KUKA KRL program: hmi.src, hmi.dat

--- hmi.src ---
&ACCESS RVO
&REL 6
&PARAM EDITMASK = *
&PARAM TEMPLATE = C:\KRC\Roboter\Template\ExpertVorgabe
DEF hmi( )
wait sec 1000
END

--- hmi.dat ---
&ACCESS RVO
&REL 6
&PARAM EDITMASK = *
&PARAM TEMPLATE = C:\KRC\Roboter\Template\ExpertVorgabe
DEFDAT hmi PUBLIC

ENDDAT
